Universal Robots URScript: d_to_c.script

def d_to_c():
  global _hidden_verificationVariable=0
  step_count_c7eae8a0_68e0_4ef2_9947_bb0ba24c3e4e = 0.0
  thread Step_Counter_Thread_9af9f7b9_c5ac_40c2_829e_f99cfe165897():
    while (True):
      step_count_c7eae8a0_68e0_4ef2_9947_bb0ba24c3e4e = step_count_c7eae8a0_68e0_4ef2_9947_bb0ba24c3e4e + 1.0
      sync()
    end
  end
  run Step_Counter_Thread_9af9f7b9_c5ac_40c2_829e_f99cfe165897()
  set_gravity([0.0, 0.0, 9.82])
  set_safety_mode_transition_hardness(1)
  set_tool_communication(False, 115200, 0, 1, 1.5, 3.5)
  set_tool_output_mode(0)
  set_tool_digital_output_mode(0, 1)
  set_tool_digital_output_mode(1, 1)
  set_tool_voltage(0)
  set_tcp(p[0.028210348281514253,-0.09610723587300697,-0.09969041498611403,0.0,0.0,0.0])
  set_standard_analog_input_domain(0, 1)
  set_standard_analog_input_domain(1, 1)
  set_tool_analog_input_domain(0, 1)
  set_tool_analog_input_domain(1, 1)
  set_analog_outputdomain(0, 0)
  set_analog_outputdomain(1, 0)
  set_input_actions_to_default()
  set_target_payload(0.260000, [0.050000, -0.008000, 0.024000], [0.000163, 0.000163, 0.000163, 0.000000, 0.000000, 0.000000])
  global Plane_1=p[0.32571614183608727,0.7933870146316717,0.11820742021636722,-2.208244884171713,-0.24738609815952348,-1.9195085473101943]
  global Plane_2=p[0.3436052139151623,0.7478032414335104,0.10077839665899768,2.768545736097797,0.1284831553507919,1.3672805628273381]
  global Plane_3=p[0.31945151854627996,0.6757990361168175,0.09459088830114093,2.7301760593116526,-0.049483824131046385,1.4252239353300047]
  global Plane_4=p[0.3372257363094211,0.6222230974198586,0.07001667903587716,2.621672423508307,-0.12240385890263918,1.4373011913128484]
  # begin: URCap Installation Node
  #   Source: External Control, 1.0.5, FZI Research Center for Information Technology
  #   Type: External Control
  # end: URCap Installation Node
  global Waypoint_2_from_p=p[.316087251829, .723602915222, .117785948188, -1.534897116856, -2.238580377483, 1.127488613076]
  global Waypoint_2_to_p=p[.245285302051, .570707986784, .053284895193, -1.842505813067, -1.391815245909, .068652086003]
  global Waypoint_1_from_p=p[.337282996076, .452563611337, .146255332642, -1.608315379440, -2.197770377912, 1.042923882249]
  global Waypoint_1_to_p=p[.195289857698, .411467596061, .021274690011, -1.734256890751, -1.516878110441, .432059224907]
  global Waypoint_3_from_p=p[.340786884756, .238628334100, .127315808714, -1.537384367056, -2.122233192013, 1.086388726493]
  global Waypoint_3_to_p=p[.152628280686, .275821245204, -.005995417926, -1.612115076189, -1.600774559356, .740435210172]
  while (True):
    $ 2 "Robot Program"
    $ 3 "bow_section≔-1"
    global bow_section=-1
    $ 4 "If bow_section≟-1"
    if (bow_section == -1):
      $ 5 "MoveJ"
      $ 6 "Waypoint_2" "breakAfter"
      movej(pose_add(get_target_tcp_pose(), pose_sub(Waypoint_2_to_p, Waypoint_2_from_p)), a=1.3962634015954636, v=1.0471975511965976)
    else:
      $ 7 "ElseIf bow_section≟0"
      if (bow_section == 0):
        $ 8 "MoveJ"
        $ 9 "Waypoint_1" "breakAfter"
        movej(pose_add(get_target_tcp_pose(), pose_sub(Waypoint_1_to_p, Waypoint_1_from_p)), a=1.3962634015954636, v=1.0471975511965976)
      else:
        $ 10 "Else" "noBreak"
        $ 11 "MoveJ"
        $ 12 "Waypoint_3" "breakAfter"
        movej(pose_add(get_target_tcp_pose(), pose_sub(Waypoint_3_to_p, Waypoint_3_from_p)), a=1.3962634015954636, v=1.0471975511965976)
      end
    end
  end
end
